// TIA Portal V19 export
FUNCTION "RD_Done" : Bool   // FC170, LAD
// stored: SetENOAutomatically false
   VAR_INPUT
      op : Date_And_Time;
   END_VAR
   VAR_TEMP
      PIPPO : Bool;
   END_VAR
BEGIN

REGION Network 1 (SCL)
   // 
   #RD_Done := DATE_TO_INT(DT_TO_DATE(#op)) <> 0;
   ENO := #RD_Done;
END_REGION
END_FUNCTION
